# EPICS IOC start-up script: iocsh/ethercatmcGenericStatusWord.iocsh
ethercatmcCreateAsynParam $(MOTOR_PORT) $(PARAM_NAME)        UInt32Digital

ethercatmcCreateAsynParam $(MOTOR_PORT) $(PARAM_NAME)_NamBit0   Octet
ethercatmcCreateAsynParam $(MOTOR_PORT) $(PARAM_NAME)_NamBit1   Octet
ethercatmcCreateAsynParam $(MOTOR_PORT) $(PARAM_NAME)_NamBit2   Octet
ethercatmcCreateAsynParam $(MOTOR_PORT) $(PARAM_NAME)_NamBit3   Octet
ethercatmcCreateAsynParam $(MOTOR_PORT) $(PARAM_NAME)_NamBit4   Octet
ethercatmcCreateAsynParam $(MOTOR_PORT) $(PARAM_NAME)_NamBit5   Octet
ethercatmcCreateAsynParam $(MOTOR_PORT) $(PARAM_NAME)_NamBit6   Octet
ethercatmcCreateAsynParam $(MOTOR_PORT) $(PARAM_NAME)_NamBit7   Octet
ethercatmcCreateAsynParam $(MOTOR_PORT) $(PARAM_NAME)_NamBit8   Octet
ethercatmcCreateAsynParam $(MOTOR_PORT) $(PARAM_NAME)_NamBit9   Octet
ethercatmcCreateAsynParam $(MOTOR_PORT) $(PARAM_NAME)_NamBit10  Octet
ethercatmcCreateAsynParam $(MOTOR_PORT) $(PARAM_NAME)_NamBit11  Octet
ethercatmcCreateAsynParam $(MOTOR_PORT) $(PARAM_NAME)_NamBit12  Octet
ethercatmcCreateAsynParam $(MOTOR_PORT) $(PARAM_NAME)_NamBit13  Octet
ethercatmcCreateAsynParam $(MOTOR_PORT) $(PARAM_NAME)_NamBit14  Octet
ethercatmcCreateAsynParam $(MOTOR_PORT) $(PARAM_NAME)_NamBit15  Octet
ethercatmcCreateAsynParam $(MOTOR_PORT) $(PARAM_NAME)_NamBit16  Octet
ethercatmcCreateAsynParam $(MOTOR_PORT) $(PARAM_NAME)_NamBit17  Octet
ethercatmcCreateAsynParam $(MOTOR_PORT) $(PARAM_NAME)_NamBit18  Octet
ethercatmcCreateAsynParam $(MOTOR_PORT) $(PARAM_NAME)_NamBit19  Octet
ethercatmcCreateAsynParam $(MOTOR_PORT) $(PARAM_NAME)_NamBit20  Octet
ethercatmcCreateAsynParam $(MOTOR_PORT) $(PARAM_NAME)_NamBit21  Octet
ethercatmcCreateAsynParam $(MOTOR_PORT) $(PARAM_NAME)_NamBit22  Octet
ethercatmcCreateAsynParam $(MOTOR_PORT) $(PARAM_NAME)_NamBit23  Octet

dbLoadRecords("ethercatmcGenericStatusWord.template", "P=$(P), R=$(R), MOTOR_PORT=$(MOTOR_PORT), PARAM_NAME=$(PARAM_NAME), AXIS_NO=$(AXIS_NO=0), DESC=$(DESC)")
